PROGRAM ModoAutomatico
VAR_INPUT
	bOrdenMarcha: BOOL;
	bSimular:BOOL:=TRUE;
	goHome:BOOL := False;
	ordenHome:bool;
END_VAR
VAR_OUTPUT
	bFinCiclo:BOOL :=FALSE;
	EstadoPrensa: EstadosPrensa;
	estadohome: estadoshome;
	
END_VAR
VAR
	//Evolucion
	FlancoMarcha: R_trig;
	TemporizadorPrensado: Ton;
	
	//Simulacion
	TemporizadorSimulacion: TON;
	TempoSimulacion: TIME;
	ForzarErro: BOOL:=FALSE; //Esta variable permitirá forzar un erro de TimeOut
	MC_SetPosition_eje1:mc_setposition;
	MC_SetPosition_eje2:mc_setposition;
END_VAR

IF gohome THEN
	vueltacasa();
END_IF
IF NOT gohome THEN
	EvolucionEstados_Transicions();
	ActivacionActuacions_Lugares();
END_IF
IF bSimular THEN
	SimulacionAutomatico();
	simulacionejes();
END_IF

ACTION ActivacionActuacions_Lugares:
mover1:=FALSE;
mover2:=FALSE;

CASE EstadoPrensa OF
	EstadosPrensa.Entrando:
		posicion1:=1000;
		mover1:=TRUE;
	EstadosPrensa.Prensando:
		posicion2:=1000;
		mover2:=TRUE;
	EstadosPrensa.Liberando:
		posicion2:=0;
		mover2:=TRUE;
	EstadosPrensa.Sacando:
		posicion1:=0;
		mover1:=TRUE;
END_CASE
END_ACTION

ACTION EvolucionEstados_Transicions:
FlancoMarcha(clk:=bOrdenMarcha);
TemporizadorPrensado(in:=EstadoPrensa=EstadosPrensa.Aguantando, PT:=T#3S);
CASE EstadoPrensa OF
	EstadosPrensa.Parada:
		IF flancomarcha.Q THEN
			EstadoPrensa:=EstadosPrensa.Entrando;
		END_IF
	EstadosPrensa.Entrando:
		IF controlejes.MC_MoveAbsolute_eje1.Done THEN
			EstadoPrensa:=EstadosPrensa.Prensando;
		END_IF
	EstadosPrensa.Prensando:
		IF controlejes.MC_MoveAbsolute_eje2.Done THEN
			EstadoPrensa:=EstadosPrensa.Aguantando;
		END_IF
	EstadosPrensa.Aguantando:
		IF TemporizadorPrensado.Q THEN
			EstadoPrensa:=EstadosPrensa.Liberando;
		END_IF
	EstadosPrensa.Liberando:
		IF controlejes.MC_MoveAbsolute_eje2.Done THEN
			EstadoPrensa:=EstadosPrensa.Sacando;
		END_IF
	EstadosPrensa.Sacando:
		IF controlejes.MC_MoveAbsolute_eje1.Done THEN
			EstadoPrensa:=EstadosPrensa.Parada;
			bFinCiclo:=TRUE;
		END_IF
END_CASE
END_ACTION

ACTION SimulacionAutomatico:
//Se estamos simulando o pulsador1 activará ambos pulsadores
io.Pulsador2:=IO.Pulsador1;
TemporizadorSimulacion(IN:=TRUE, PT:=TempoSimulacion);
MC_SetPosition_eje1.execute:=FALSE;
MC_SetPosition_eje2.execute:=FALSE;

CASE EstadoPrensa OF
	EstadosPrensa.Parada:
		TemporizadorSimulacion(IN:=FALSE);
		TempoSimulacion:=T#5S;
		
	EstadosPrensa.Entrando:
		IF TemporizadorSimulacion.Q THEN
			MC_SetPosition_eje1.position:=1000;
			MC_SetPosition_eje1.execute:=TRUE;
			TemporizadorSimulacion(IN:=FALSE);
			TempoSimulacion:=T#2S;
		END_IF
	EstadosPrensa.Prensando:
		IF TemporizadorSimulacion.Q THEN
			MC_SetPosition_eje2.position:=1000;
			MC_SetPosition_eje2.execute:=TRUE;
			TemporizadorSimulacion(IN:=FALSE);
			TempoSimulacion:=T#3S;
		END_IF
	EstadosPrensa.Aguantando:
		TemporizadorSimulacion(IN:=FALSE);
	EstadosPrensa.Liberando:
		IF TemporizadorSimulacion.Q THEN
			MC_SetPosition_eje2.position:=0;
			MC_SetPosition_eje2.execute:=TRUE;
			TemporizadorSimulacion(IN:=FALSE);
			TempoSimulacion:=T#2S;
		END_IF
	EstadosPrensa.Sacando:
		IF TemporizadorSimulacion.Q THEN
			MC_SetPosition_eje1.position:=0;
			MC_SetPosition_eje1.execute:=TRUE;
			TemporizadorSimulacion(IN:=FALSE);
			TempoSimulacion:=T#5S;
		END_IF
END_CASE
//Se queremos forzar un erro metemoslle un minuto o temporizador
IF ForzarErro THEN
	TempoSimulacion:= T#1M;
END_IF
END_ACTION

ACTION simulacionEjes:
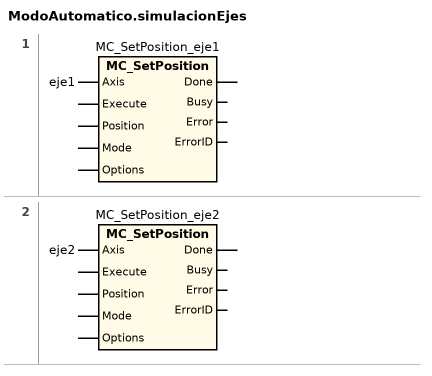
// NETWORK 1
MC_SetPosition_eje1(Axis := eje1); // MC_SetPosition

// NETWORK 2
MC_SetPosition_eje2(Axis := eje2); // MC_SetPosition
END_ACTION

ACTION vueltacasa:
mover1:=FALSE;
mover2:=FALSE;

CASE estadohome OF
	estadoshome.espera:
		IF gohome THEN
			estadohome:= estadoshome.subiendo;
		END_IF
	estadoshome.subiendo:
		posicion2:=0;
		mover2:=TRUE;
		IF controlejes.MC_MoveAbsolute_eje2.Done THEN
			estadohome:= estadoshome.sacando;
		END_IF
	estadoshome.sacando:
		posicion1:=0;
		mover1:=TRUE;
		IF controlejes.MC_MoveAbsolute_eje1.Done THEN
			estadohome:= estadoshome.ok;
		END_IF
	estadoshome.ok:
		estadohome:= estadoshome.espera;
		gohome:=FALSE;
END_CASE
END_ACTION

END_PROGRAM

(* stored: Version 1.1.0.1, ProductVersion 3.1.4024.9
   POU ModoAutomatico: Id {6eceedba-4990-4fd6-8512-9186e357f675}, SpecialFunc None
   Action ActivacionActuacions_Lugares: Id {ae29a4a6-c628-4f85-9089-745eb4b4cf59}
   Action EvolucionEstados_Transicions: Id {5708452f-5076-4b64-8388-a276cdf281ad}
   Action SimulacionAutomatico: Id {f4626de2-3467-4248-a01d-b0d66739e1c0}
   Action simulacionEjes: Id {fd16b832-b3d5-45b3-8fde-61e7176bd2fe}
   Action vueltacasa: Id {29aa0a76-c7d5-4a19-8f04-bc0937bc62ff} *)
